PROGRAM MAIN
VAR
    fbSepSol1  : FB_SolSpringPiston_2Pos;
    fbSepSol2  : FB_SolSpringPiston_2Pos;
    fbSepSol3  : FB_SolSpringPiston_2Pos;
    fbPushSol1 : FB_SolSpringPiston_2Pos;
    fbPushSol2 : FB_SolSpringPiston_2Pos;
    fbPushSol3 : FB_SolSpringPiston_2Pos;
    fbGripSolL : FB_SolSpringPiston_2Pos;
    fbGripSolR : FB_SolSpringPiston_2Pos;

    // Full-machine sequencer coordinating the 3 pairs of (SepSolN,
    // PushSolN) + the 2 grip pistons. In this panel solution the master
    // cycle is the ONLY auto driver — the per-piston auto tiles
    // (bench-only feature) are removed, so no OR-merge at the call sites.
    fbMasterAutoCycle : FB_MasterAutoCycle;

    // Robot TCP/IP client — TCP-only protocol on :6001. Carries tuning
    // params + New_Bulb + STATE/CMD (state push out, command in). The
    // former discrete-I/O handshake (STAND_SEQ_DO/DI) is retired.
    fbRobotTcp : FB_RobotTcpClient;

    // Robot TCP command channel (nRobotCmd: 0=none, 1=start cycle,
    // 2=reset error). Consumed as a LEVEL and cleared on consumption --
    // see the body for why edge-detecting it deadlocked the machine.
    // bRobotStartPulse is the resulting one-scan pulse handed to
    // fbMasterAutoCycle's bExtStartPulse.
    bRobotStartPulse : BOOL;

    // PB3 rising edge in Auto is the operator START: "home the pistons and arm
    // the machine". Drives stMasterAuto.bStart, the same field as the HMI
    // button. PB3 because it is the GREEN button (PB1 red, PB2 orange) and this
    // is the go-ahead; it used to be PB1.
    //
    // Note it drives bStart, NOT bSimStartAssembly. Under the arming model
    // START no longer runs a bulb cycle, and bSimStartAssembly keeps its own
    // distinct job as the bench stand-in for the robot's CMD:1.
    fbTrigPb3 : R_TRIG;

    // PB2 rising edge in Auto -- RESET, but only while latched in ERR.
    fbTrigPb2 : R_TRIG;

    // The two Automatic HOLD gestures (2026-08-05). Each TON's IN is the
    // gesture itself, so releasing the button resets the elapsed time; .Q is a
    // level, so each is edge-detected to fire once per press.
    //
    //   PB1 held  -> STOP (disarm to NOT_HOMED)
    //   PB2 + PB3 -> run one bulb from IDLE, the operator's parallel to CMD:1
    //
    // Durations come from GVL_HmiPersistent.stMasterAutoCfg so they are tunable
    // on AutoMain without a rebuild.
    tonPb1Stop    : TON;
    fbTrigPb1Stop : R_TRIG;
    tonPbCombo    : TON;
    fbTrigPbCombo : R_TRIG;

    // One-scan pulse from the PB2+PB3 combo, OR-merged with the robot's start
    // pulse into fbMasterAutoCycle.bExtStartPulse -- both mean "run one bulb".
    bComboStartPulse : BOOL;

    // Scratch copies of the global machine mode, computed once per scan and
    // fanned out to all eight pistons (both eMode and bMode) just below.
    bMachineAuto : BOOL;
    bManualMode  : BOOL;   // = NOT bMachineAuto; gates PB jogs
    eMachineMode : E_ControlMode;

    // Flushes GVL_HmiPersistent to disk once the operator stops editing.
    // PERSISTENT alone never wrote anything on a power cut -- see the FB
    // header. Called last so it sees this scan's final config values.
    fbPersistentSave : FB_PersistentAutoSave;

    // THROWAWAY -- Phase 0 gate of docs/plans/log-csv-file.md. Idle until an
    // operator sets GVL_Log.bLogFileProbeRun, so it costs one CASE test per
    // scan and nothing else. DELETE with the FB once the probe has answered
    // whether WinCE 7 ARM can do file I/O and which path is writable.
    fbLogFileSpike : FB_LogFileSpike;

    // Status-lamp blink source. A self-resetting TON toggling a BOOL gives a
    // 50% duty cycle; the TON on its own only produces a one-scan pulse,
    // which would make the lamp flicker rather than blink.
    tonBlink : TON;
    bBlink   : BOOL;

    // Wall clock for the log timestamps. Lives here because F_LogEvent is a
    // FUNCTION and cannot own an FB instance. dwCycle is in SECONDS.
    fbLocalTime : Tc2_Utilities.FB_LocalSystemTime;
    nLastSec    : WORD := 16#FFFF;   // impossible value, forces a first build
    sHH, sMM, sSS : STRING(2);
END_VAR

(* ==========================================
   0. CONTINUOUS IS DISABLED ON THE REAL MACHINE
   Forced FALSE every scan, not merely cleared at boot. The production
   machine never free-runs: every cycle is started by the operator or by the
   robot's CMD:1. The checkbox was removed from AutoMain, but a VISU page is
   only one of several writers — FlowerPyHmi has its own Continuous checkbox
   on two pages and reaches the field over ADS — so the field itself has to
   be the enforcement point. Any write is overwritten within one scan.

   It USED to be load-bearing: the IDLE branch tested it as a level, so a TRUE
   here re-armed a cycle with nothing external gating it. That is no longer the
   case -- the arming-model change of 2026-07-29 removed it from IDLE's exit
   condition, and the FB now writes bContinuous ten times and reads it ZERO
   times. This force-clear is belt-and-braces, not the interlock. What actually
   prevents power-up motion is eStep's NOT_HOMED default, below.

   bAutoMode is deliberately NOT touched (operator decision, 2026-07-27): the
   panel comes back in Automatic after a power cycle, still needing a real
   start trigger.

   This block used to add that it therefore came back in IDLE reporting
   nStateOut = 0, so "a robot already running may request a cycle straight
   after power-up -- that is the intended production behaviour". SUPERSEDED
   2026-07-29 and no longer true in either half. stHmi.eStep now DEFAULTS to
   NOT_HOMED (40), and GVL_HMI is plain VAR_GLOBAL so that initialiser is
   re-applied on every cold boot and download. A persisted bAutoMode = TRUE
   brings the panel back in Automatic but UN-ARMED, reporting 40, which the
   robot answers CMD:0 (wait). An operator START is required before anything
   can move. bAutoMode persists; the arming does not. See the ARMING MODEL
   section in CLAUDE.md.

   The timers, bNoSensors and bBypassPlateSensors are untouched too — they
   are operator config and persisting them is the point of the flush.
   ========================================== *)

(* ==========================================
   0a. LOG WALL CLOCK
   Refreshes GVL_Log.sNow, which F_LogEvent stamps into every entry so the
   Logs page can show a Time column. Rebuilt only when the second actually
   rolls over — the string work is trivial but there is no reason to redo it
   100 times a second.

   bValid gates it: an unset RTC shows '--:--:--' rather than a plausible
   wrong time, which is the difference between "the clock is not set" and
   "these events happened at 00:00:03".
   ========================================== *)
fbLocalTime(bEnable := TRUE, dwCycle := 1);

IF NOT fbLocalTime.bValid THEN
    GVL_Log.sNow := '--:--:--';
ELSIF fbLocalTime.systemTime.wSecond <> nLastSec THEN
    nLastSec := fbLocalTime.systemTime.wSecond;
    // RIGHT(CONCAT('0', n), 2) is the zero-pad: '7' -> '07', '17' -> '17'.
    sHH := RIGHT(CONCAT('0', WORD_TO_STRING(fbLocalTime.systemTime.wHour)), 2);
    sMM := RIGHT(CONCAT('0', WORD_TO_STRING(fbLocalTime.systemTime.wMinute)), 2);
    sSS := RIGHT(CONCAT('0', WORD_TO_STRING(fbLocalTime.systemTime.wSecond)), 2);
    GVL_Log.sNow := CONCAT(CONCAT(CONCAT(CONCAT(sHH, ':'), sMM), ':'), sSS);
END_IF

(* ==========================================
   Master auto-cycle — coordinates the 3 pairs of (Sep,Push) pistons
   with the robot handshake. Called BEFORE the per-piston
   auto FBs and BEFORE the piston FBs so its bSepCmd* / bPushCmd*
   outputs feed forward this scan.
   Master reads bIs* from the piston stHmi structs — those carry the
   previous scan's values (100 µs lag, negligible for a physical
   machine).
   ========================================== *)
fbMasterAutoCycle.bSepIsExtended[1]   := GVL_HMI.stSepSol1.bIsExtended;
fbMasterAutoCycle.bSepIsExtended[2]   := GVL_HMI.stSepSol2.bIsExtended;
fbMasterAutoCycle.bSepIsExtended[3]   := GVL_HMI.stSepSol3.bIsExtended;
fbMasterAutoCycle.bSepIsRetracted[1]  := GVL_HMI.stSepSol1.bIsRetracted;
fbMasterAutoCycle.bSepIsRetracted[2]  := GVL_HMI.stSepSol2.bIsRetracted;
fbMasterAutoCycle.bSepIsRetracted[3]  := GVL_HMI.stSepSol3.bIsRetracted;
fbMasterAutoCycle.bPushIsExtended[1]  := GVL_HMI.stPushSol1.bIsExtended;
fbMasterAutoCycle.bPushIsExtended[2]  := GVL_HMI.stPushSol2.bIsExtended;
fbMasterAutoCycle.bPushIsExtended[3]  := GVL_HMI.stPushSol3.bIsExtended;
fbMasterAutoCycle.bPushIsRetracted[1] := GVL_HMI.stPushSol1.bIsRetracted;
fbMasterAutoCycle.bPushIsRetracted[2] := GVL_HMI.stPushSol2.bIsRetracted;
fbMasterAutoCycle.bPushIsRetracted[3] := GVL_HMI.stPushSol3.bIsRetracted;

(* Grip pistons — L=[1], R=[2]. *)
fbMasterAutoCycle.bGripIsExtended[1]  := GVL_HMI.stGripSolL.bIsExtended;
fbMasterAutoCycle.bGripIsExtended[2]  := GVL_HMI.stGripSolR.bIsExtended;
fbMasterAutoCycle.bGripIsRetracted[1] := GVL_HMI.stGripSolL.bIsRetracted;
fbMasterAutoCycle.bGripIsRetracted[2] := GVL_HMI.stGripSolR.bIsRetracted;

(* Plate-presence sensors gate the cycle at WAIT_PLATE. Wire the raw
   GVL_App copies straight into the master cycle. Also mirror them onto
   GVL_HMI so the classic VISU / web HMI indicator lamps can bind. *)
fbMasterAutoCycle.bPlateSenL := GVL_App.bPlateSenL;
fbMasterAutoCycle.bPlateSenR := GVL_App.bPlateSenR;
GVL_HMI.bPlateSenL := GVL_App.bPlateSenL;
GVL_HMI.bPlateSenR := GVL_App.bPlateSenR;

(* ==========================================
   ROBOT COMMAND CONSUMPTION (nRobotCmd, written by fbRobotTcp on each
   CMD:<n> reply -- see the fbRobotTcp call further down).

   Consumed as a LEVEL and CLEARED here. The PLC clearing the field is the
   acknowledgement; the robot zeroing it after the next state push is now
   belt-and-braces rather than load-bearing.

   This used to be a pair of R_TRIGs on nRobotCmd = 1 / = 2, and nothing on
   the PLC side ever reset the field. That deadlocked the machine
   (2026-07-28, found on the real machine): a CMD:1 arriving while the panel
   was in Manual or latched in ERR fired the edge, the FB's IDLE branch
   correctly refused it, and nRobotCmd stayed at 1 forever. The robot
   re-asserts CMD:1 in every STATE reply until it sees the panel leave IDLE
   -- but re-sending a value that is already 1 produces no rising edge. So
   the robot waited for a state change while the PLC waited for an edge that
   could never come, and the Robot page showed CMD:1 arriving happily the
   whole time.

   Clearing makes it self-healing. A request that cannot be honoured this
   scan is dropped, and the robot's next keep-alive re-asserts it ~1 s
   later. Repeat pulses are harmless: only FB_MasterAutoCycle's IDLE branch
   consumes bExtStartPulse, and it is gated on bMachineAuto.

   Diagnostic note: nRobotCmd now reads 0 almost always, because it is
   consumed within a scan of arriving. The trace of a robot start is the
   'External start pulse' entry on the Logs page, and stRobot.sLastMessage
   still shows the raw CMD frame.

   RESET is fanned into the HMI bReset flag so operator- and robot-initiated
   resets share one consumption path inside the FB.
   ========================================== *)
bRobotStartPulse := FALSE;

IF GVL_Robot.stParams.nRobotCmd = 1 THEN
    bRobotStartPulse             := TRUE;
    GVL_Robot.stParams.nRobotCmd := 0;
ELSIF GVL_Robot.stParams.nRobotCmd = 2 THEN
    GVL_HMI.stMasterAuto.bReset  := TRUE;
    GVL_Robot.stParams.nRobotCmd := 0;
END_IF

fbMasterAutoCycle(
    bExtStartPulse := bRobotStartPulse OR bComboStartPulse,
    bMachineAuto   := GVL_HMI.bAutoMode,
    stHmi          := GVL_HMI.stMasterAuto,
    stCfg          := GVL_HmiPersistent.stMasterAutoCfg,
    stRobot        := GVL_Robot.stRobot
);

(* Global Auto/Manual hard interlock. The machine-wide bAutoMode is the single
   source of truth for every piston's mode — driven unconditionally each scan
   onto BOTH eMode and bMode so a per-piston toggle cannot create a second
   control path (no double-control). FB_SolSpringPiston_2Pos edge-syncs
   bMode<->eMode, so forcing only one would let a stray toggle propagate for a
   scan; forcing both closes that gap. In Automatic the master cycle owns all
   six pistons; in Manual the operator jogs them and the cycle is held in IDLE. *)
bMachineAuto := GVL_HMI.bAutoMode;
eMachineMode := SEL(bMachineAuto, E_ControlMode.Manual, E_ControlMode.Automatic);
GVL_HMI.stSepSol1.eMode  := eMachineMode;  GVL_HMI.stSepSol1.bMode  := bMachineAuto;
GVL_HMI.stPushSol1.eMode := eMachineMode;  GVL_HMI.stPushSol1.bMode := bMachineAuto;
GVL_HMI.stSepSol2.eMode  := eMachineMode;  GVL_HMI.stSepSol2.bMode  := bMachineAuto;
GVL_HMI.stPushSol2.eMode := eMachineMode;  GVL_HMI.stPushSol2.bMode := bMachineAuto;
GVL_HMI.stSepSol3.eMode  := eMachineMode;  GVL_HMI.stSepSol3.bMode  := bMachineAuto;
GVL_HMI.stPushSol3.eMode := eMachineMode;  GVL_HMI.stPushSol3.bMode := bMachineAuto;
GVL_HMI.stGripSolL.eMode := eMachineMode;  GVL_HMI.stGripSolL.bMode := bMachineAuto;
GVL_HMI.stGripSolR.eMode := eMachineMode;  GVL_HMI.stGripSolR.bMode := bMachineAuto;

(* ==========================================
   Panel push buttons. PB1 is RED, PB2 ORANGE, PB3 GREEN, and the colours
   drive the assignment.

   IN MANUAL — all three are momentary jogs. Hold to extend, release to
   retract: PB1 grip, PB2 Sep, PB3 Push. Unchanged.

   IN AUTOMATIC — three operator gestures, no jogs at all (operator decision
   2026-08-05: manual moves belong in Manual mode, not in any Auto state):

   * PB1 (red), HELD for tPbStopHoldMs   -> STOP. Disarms to NOT_HOMED.
   * PB3 (green), rising edge            -> START. "Home the pistons and arm."
                                            Drives stMasterAuto.bStart, the
                                            same field as the HMI button.
   * PB2 + PB3 together, HELD for
     tPbStartHoldMs, from IDLE           -> run ONE bulb cycle. The operator's
                                            parallel to the robot's CMD:1.
   * PB2 (orange), rising edge, in ERR   -> RESET.

   Why the two multi-second holds: both are consequential (one stops the
   machine, one starts a bulb), and a hold cannot be triggered by a knock or a
   brushed sleeve the way an edge can. Durations are operator-tunable on
   AutoMain rather than compiled in.

   PB3-vs-combo disambiguation: the standalone START edge is suppressed while
   PB2 is pressed, so the combo does not fire START on the way in. Press ORANGE
   first, then GREEN.

   Green-first is NOT harmless, and it was measured rather than assumed. It
   fires a plain START, so the machine re-homes. bComboStartPulse is one scan
   and bExtStartPulse is consumed ONLY by the IDLE branch, so:
     - homing done inside the hold  -> pointless re-home, then the cycle runs
     - still homing when it expires -> pulse DROPPED, no cycle, and the R_TRIG
                                       will not re-offer it while held
   On the machine, with real strokes, the second is the case to expect. See the
   TODO in CLAUDE.md about latching the request instead of pulsing it.

   * LED1 mirrors the press, and BLINKS while the STOP hold is counting.
   * LED2 mirrors the press.
   * LED3 is a state prompt in Auto -- assigned further down, after bBlink.
   ========================================== *)
GVL_App.bLedPb2 := GVL_App.bPb2;
(* PB3's LED is no longer a press mirror in Auto -- it is the "press me to arm"
   prompt. Assigned further down, after bBlink is refreshed, so the blink is
   this scan's value rather than last scan's. *)

(* ==========================================
   Machine status lamps (DO 12 green / DO 13 red).
   Unlike the PB LEDs above, which are dumb press mirrors, these report
   machine state:

     RED   = the master cycle is in its latched ERR state.
     GREEN = Auto and IDLE        -> steady  (armed, waiting for a start)
             Auto and cycling     -> blink   (running)
             Manual, or in ERR    -> off

   Green is off in ERR so the two lamps never contradict each other: red on
   with green also lit would read as "faulted but running". Green is off in
   Manual because it means "the automatic cycle is live", which is precisely
   what Manual is not.

   Blink source is a self-resetting TON toggling bBlink, giving 400 ms on /
   400 ms off. Using tonBlink.Q directly would light the lamp for a single
   scan per period -- invisible.
   ========================================== *)
tonBlink(IN := NOT tonBlink.Q, PT := T#400MS);
IF tonBlink.Q THEN
    bBlink := NOT bBlink;
END_IF

GVL_App.bLedRed := (GVL_HMI.stMasterAuto.eStep = E_MasterAutoStep.ERR);

IF NOT bMachineAuto
   OR GVL_HMI.stMasterAuto.eStep = E_MasterAutoStep.ERR
   OR GVL_HMI.stMasterAuto.eStep = E_MasterAutoStep.NOT_HOMED THEN
    (* Off in NOT_HOMED as well as Manual/ERR: green means "the automatic cycle
       is live and armed", and an un-homed machine is precisely not that. PB3's
       own green LED is the "press me" signal in that state, so the two are not
       competing for the operator's attention. *)
    GVL_App.bLedGreen := FALSE;
ELSIF GVL_HMI.stMasterAuto.eStep = E_MasterAutoStep.IDLE THEN
    GVL_App.bLedGreen := TRUE;
ELSE
    GVL_App.bLedGreen := bBlink;
END_IF

(* ==========================================
   PANEL GESTURES IN AUTOMATIC
   fbMasterAutoCycle already ran this scan, so eStep is current here.

   Both hold timers are driven with IN := <gesture held AND in Auto>, so
   releasing the button -- or leaving Auto -- resets the elapsed time and the
   operator has to start the hold again. .Q is a LEVEL, true for as long as the
   hold persists, so each one is edge-detected to fire exactly once per press.
   ========================================== *)

(* --- PB1 held -> STOP ------------------------------------------------------
   Writes stMasterAuto.bStop, the same field as the HMI STOP button, so the FB's
   existing Section 2 override handles it: disarm to NOT_HOMED, no error code. *)
tonPb1Stop(IN := bMachineAuto AND GVL_App.bPb1,
           PT := UDINT_TO_TIME(GVL_HmiPersistent.stMasterAutoCfg.tPbStopHoldMs));
fbTrigPb1Stop(CLK := tonPb1Stop.Q);
IF fbTrigPb1Stop.Q THEN
    GVL_HMI.stMasterAuto.bStop := TRUE;
END_IF;

(* --- PB2 + PB3 held -> run one bulb ----------------------------------------
   Fed into the SAME bExtStartPulse input the robot's CMD:1 uses, because it
   means exactly the same thing: "run one bulb". The FB's IDLE branch is the
   only consumer, and it is gated on bMachineAuto, so this cannot start a cycle
   from NOT_HOMED or from ERR -- the arming model is untouched. *)
tonPbCombo(IN := bMachineAuto AND GVL_App.bPb2 AND GVL_App.bPb3,
           PT := UDINT_TO_TIME(GVL_HmiPersistent.stMasterAutoCfg.tPbStartHoldMs));
fbTrigPbCombo(CLK := tonPbCombo.Q);
bComboStartPulse := fbTrigPbCombo.Q;
IF bComboStartPulse THEN
    F_LogEvent(eSev := E_LogSev.INFO, sSource := 'MAIN',
               sMsg := 'PB2+PB3 held: operator bulb start');
END_IF;

(* --- PB2 in ERR -> RESET ---------------------------------------------------
   An edge, not a hold: the machine is already stopped and latched, so there is
   nothing for a stray press to interrupt. Writes the same bReset field as the
   HMI button and the robot's CMD:2. *)
fbTrigPb2(CLK := GVL_App.bPb2);
IF bMachineAuto AND fbTrigPb2.Q
   AND GVL_HMI.stMasterAuto.eStep = E_MasterAutoStep.ERR THEN
    GVL_HMI.stMasterAuto.bReset := TRUE;
END_IF;

(* --- PB1 LED: press mirror, blinking while the STOP hold counts ------------
   A hold-to-act button with no feedback is guesswork; the blink tells the
   operator the hold is being counted. Assigned after bBlink is refreshed so it
   is this scan's value. *)
IF bMachineAuto AND GVL_App.bPb1 AND NOT tonPb1Stop.Q THEN
    GVL_App.bLedPb1 := bBlink;
ELSE
    GVL_App.bLedPb1 := GVL_App.bPb1;
END_IF

(* --- PB3 LED: "press me to arm" prompt ------------------------------------
   Blinks while in Auto and un-homed, off otherwise in Auto. Falls back to a raw
   press mirror in Manual, where PB3 is the Push jog and the LED keeps its
   original wiring-diagnostic role. *)
IF bMachineAuto THEN
    GVL_App.bLedPb3 := (GVL_HMI.stMasterAuto.eStep = E_MasterAutoStep.NOT_HOMED) AND bBlink;
ELSE
    GVL_App.bLedPb3 := GVL_App.bPb3;
END_IF

(* --- PB3 edge -> START ----------------------------------------------------
   Suppressed while PB2 is pressed so the PB2+PB3 combo does not fire a START on
   its way in. Press ORANGE first, then GREEN -- green-first can silently lose
   the cycle request, see the header. *)
fbTrigPb3(CLK := GVL_App.bPb3);
IF bMachineAuto AND NOT GVL_App.bPb2 AND fbTrigPb3.Q THEN
    GVL_HMI.stMasterAuto.bStart := TRUE;
END_IF;

bManualMode := NOT bMachineAuto;

(* ==========================================
   Pin separators (SOL-Spring, 2 limit switches, single Extend coil).
   The master cycle is the only auto driver; in Manual the piston FB
   ignores bAutoCmd* and follows the operator's jog buttons instead.
   ========================================== *)
fbSepSol1(
    bAutoCmdExtend   := fbMasterAutoCycle.bSepCmdExtend[1],
    bAutoCmdRetract  := fbMasterAutoCycle.bSepCmdRetract[1],
    bJogExtend       := bManualMode AND GVL_App.bPb2,
    bSwitchExtended  := GVL_App.bSensorSepExtended1,
    bSwitchRetracted := GVL_App.bSensorSepRetracted1,
    stHmi            := GVL_HMI.stSepSol1,
    bOutSolenoid     => GVL_App.bValveSepExtend1
);

fbSepSol2(
    bAutoCmdExtend   := fbMasterAutoCycle.bSepCmdExtend[2],
    bAutoCmdRetract  := fbMasterAutoCycle.bSepCmdRetract[2],
    bJogExtend       := bManualMode AND GVL_App.bPb2,
    bSwitchExtended  := GVL_App.bSensorSepExtended2,
    bSwitchRetracted := GVL_App.bSensorSepRetracted2,
    stHmi            := GVL_HMI.stSepSol2,
    bOutSolenoid     => GVL_App.bValveSepExtend2
);

fbSepSol3(
    bAutoCmdExtend   := fbMasterAutoCycle.bSepCmdExtend[3],
    bAutoCmdRetract  := fbMasterAutoCycle.bSepCmdRetract[3],
    bJogExtend       := bManualMode AND GVL_App.bPb2,
    bSwitchExtended  := GVL_App.bSensorSepExtended3,
    bSwitchRetracted := GVL_App.bSensorSepRetracted3,
    stHmi            := GVL_HMI.stSepSol3,
    bOutSolenoid     => GVL_App.bValveSepExtend3
);

(* ==========================================
   Pin pushers
   ========================================== *)
fbPushSol1(
    bAutoCmdExtend   := fbMasterAutoCycle.bPushCmdExtend[1],
    bAutoCmdRetract  := fbMasterAutoCycle.bPushCmdRetract[1],
    bJogExtend       := bManualMode AND GVL_App.bPb3,
    bSwitchExtended  := GVL_App.bSensorPushExtended1,
    bSwitchRetracted := GVL_App.bSensorPushRetracted1,
    stHmi            := GVL_HMI.stPushSol1,
    bOutSolenoid     => GVL_App.bValvePushExtend1
);

fbPushSol2(
    bAutoCmdExtend   := fbMasterAutoCycle.bPushCmdExtend[2],
    bAutoCmdRetract  := fbMasterAutoCycle.bPushCmdRetract[2],
    bJogExtend       := bManualMode AND GVL_App.bPb3,
    bSwitchExtended  := GVL_App.bSensorPushExtended2,
    bSwitchRetracted := GVL_App.bSensorPushRetracted2,
    stHmi            := GVL_HMI.stPushSol2,
    bOutSolenoid     => GVL_App.bValvePushExtend2
);

fbPushSol3(
    bAutoCmdExtend   := fbMasterAutoCycle.bPushCmdExtend[3],
    bAutoCmdRetract  := fbMasterAutoCycle.bPushCmdRetract[3],
    bJogExtend       := bManualMode AND GVL_App.bPb3,
    bSwitchExtended  := GVL_App.bSensorPushExtended3,
    bSwitchRetracted := GVL_App.bSensorPushRetracted3,
    stHmi            := GVL_HMI.stPushSol3,
    bOutSolenoid     => GVL_App.bValvePushExtend3
);

(* ==========================================
   Grip pistons — side clamps (L=[1], R=[2]) that hold the plate placed
   by the robot for the duration of the Sep/Push cycle.
   ========================================== *)
fbGripSolL(
    bAutoCmdExtend   := fbMasterAutoCycle.bGripCmdExtend[1],
    bAutoCmdRetract  := fbMasterAutoCycle.bGripCmdRetract[1],
    bJogExtend       := bManualMode AND GVL_App.bPb1,
    bSwitchExtended  := GVL_App.bSensorGripExtendedL,
    bSwitchRetracted := GVL_App.bSensorGripRetractedL,
    stHmi            := GVL_HMI.stGripSolL,
    bOutSolenoid     => GVL_App.bValveGripExtendL
);

fbGripSolR(
    bAutoCmdExtend   := fbMasterAutoCycle.bGripCmdExtend[2],
    bAutoCmdRetract  := fbMasterAutoCycle.bGripCmdRetract[2],
    bJogExtend       := bManualMode AND GVL_App.bPb1,
    bSwitchExtended  := GVL_App.bSensorGripExtendedR,
    bSwitchRetracted := GVL_App.bSensorGripRetractedR,
    stHmi            := GVL_HMI.stGripSolR,
    bOutSolenoid     => GVL_App.bValveGripExtendR
);

(* ==========================================
   Robot TCP/IP client (TCP-only protocol, port 6001). Runs every scan;
   its internal state machine dials the robot server and auto-reconnects
   on drop. The former discrete-I/O handshake is retired -- start/reset
   commands arrive via CMD:<n> replies, PLC state pushes via STATE:<n>.

   Compute nStateOut immediately after the master cycle so any transition
   this scan is visible to the robot on the next STATE push. MANUAL(30)
   sentinel while bAutoMode=FALSE so the robot knows the panel is out of
   auto and won't issue CMD:1.
   ========================================== *)
IF NOT GVL_HMI.bAutoMode THEN
    GVL_Robot.stParams.nStateOut := INT#30;   (* MANUAL *)
ELSE
    GVL_Robot.stParams.nStateOut := TO_INT(GVL_HMI.stMasterAuto.eStep);
END_IF

fbRobotTcp(
    bEnable     := GVL_Robot.bTcpEnable,
    sRemoteHost := GVL_Robot.sRobotHost,
    nRemotePort := GVL_Robot.nRobotPort,
    stRobot     := GVL_Robot.stRobot,
    stParams    := GVL_Robot.stParams
);

(* ==========================================
   Persistent config flush. Called LAST so it compares this scan's final
   values, and after section 0 so the cold-boot clears are part of its
   baseline rather than looking like an operator edit.
   Writes ~2 s after the operator stops editing; logs each flush to
   GVL_Log (visible on the Logs page) so a failing write is not silent.
   ========================================== *)
fbPersistentSave();

(* ==========================================
   THROWAWAY -- Phase 0 file-I/O probe. See docs/plans/log-csv-file.md.
   Sits here, after the persistent flush, because that is the slot the real
   FB_LogCsvWriter will occupy in Phase 2 -- so whatever this proves about
   timing and error behaviour is proved where the writer will actually live.
   Does nothing until GVL_Log.bLogFileProbeRun goes TRUE.
   DELETE this call, the instance, the FB, ST_LogFileProbe and the GVL block
   once the gate has been answered.
   ========================================== *)
fbLogFileSpike();

END_PROGRAM

(* stored: Version 1.1.0.1, ProductVersion 3.1.4024.16
   POU MAIN: Id {14abf4a7-7840-47f5-84af-a7dedadf8c83}, SpecialFunc None *)
